(* PLC project FBD_EVOLUTION_6, Beckhoff Automation GmbH TwinCAT PLC Control 3.5.10.30 *)
(* stored: creationDateTime 2019-09-26T17:08:43.2216771, modificationDateTime 2019-09-26T17:08:43.2216771 *)

PROGRAM POU
VAR
	A: BOOL;
	B: BOOL;
	C: BOOL;
	D: BOOL;
END_VAR
  VAR  (* added by the conversion: wires and edge detectors of the diagram *)
    _EXECUTE20000000003_EN : BOOL;
  END_VAR

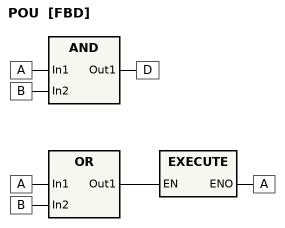
(* FBD diagram, written out as Structured Text *)
D := A AND B;
_EXECUTE20000000003_EN := A OR B;
IF _EXECUTE20000000003_EN THEN
  A := B AND C;
END_IF;
A := _EXECUTE20000000003_EN;
END_PROGRAM

CONFIGURATION Application
  RESOURCE FBD_EVOLUTION_6 ON PLC
(* global variable list GVL *)
{attribute 'qualified_only'}
VAR_GLOBAL
	IsSFCResetting : BOOL;
END_VAR
    TASK PlcTask(INTERVAL := T#0ms, PRIORITY := 20);
    PROGRAM MAIN WITH PlcTask : MAIN;
  END_RESOURCE
END_CONFIGURATION
